Universal Robots PolyScope program: motion_capture.urp

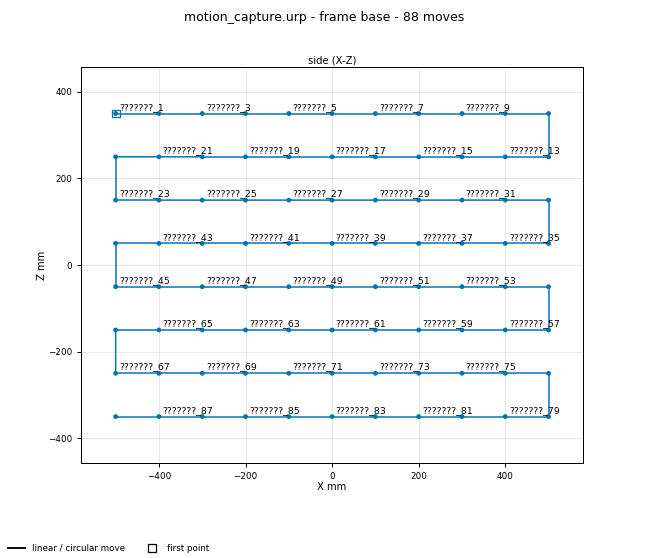
[picture p0: tool path of motion_capture.urp in frame base, 88 of 94 moves have a stored position in this frame; points joined in program order, loops and branches not executed]
Program motion_capture (installation=GD directory=/programs/GD createdIn=5.13.0 lastSavedIn=5.13.0 robotSerialNumber=20205000017)
Calibrated DH parameters: a=[-0.000157, -0.56303, -0.236706, -0.000074, -0.000109, 0]; d=[0.181705, 47.632387, 369.599619, -417.058513, 0.119878, 0.115667]; alpha=[1.570881, -0.005074, -0.001247, 1.56886, -1.570997, 0]; deltaTheta=[0, -0.405485, 5.544791, 1.143886, -0.000009, -0.000001]
InitVariablesNode
BeforeStart
  SuppressedNode
    Script file /programs/GD/ROVI/ROVI_RESET.script
      | def ROVI_RESET():
      |   if (not socket_open(host,port,socket_name)):
      |     rovi_err=902
      |     return False
      |   end
      |   socket_send_line("X0()",socket_name)
      |   ret=socket_read_line(socket_name,socket_timeout)
      |   if (ret == "OK"):
      |     rovi_err=0
      |   elif (ret == "NG"):
      |     rovi_err=to_num(socket_read_line(socket_name,socket_timeout))
      |   else:
      |     ret="NG"
      |     rovi_err=903
      |   end
      |   socket_close(socket_name)
      |   if (rovi_err != 0):
      |     if (is_popup):
      |       popup(str_cat(ret,rovi_err),title="X0",warning=True,blocking=True)
      |     end
      |     return False
      |   else:
      |     return True
      |   end
      | end
  SuppressedNode
    Script file /programs/GD/ROVI/ROVI_CAPTURE.script
      | def ROVI_CAPTURE():
      |   Y1=[0.0,0.0,0.0,0.0]
      | #  p=get_actual_tool_flange_pose()
      |   p=Bucket
      |   if (not socket_open(host,port,socket_name)):
      |     rovi_err=902
      |     return False
      |   end
      |   socket_send_string("X1(",socket_name)
      |   socket_send_string(p[0],socket_name)
      |   socket_send_string(",",socket_name)
      |   socket_send_string(p[1],socket_name)
      |   socket_send_string(",",socket_name)
      |   socket_send_string(p[2],socket_name)
      |   socket_send_string(",",socket_name)
      |   socket_send_string(p[3],socket_name)
      |   socket_send_string(",",socket_name)
      |   socket_send_string(p[4],socket_name)
      |   socket_send_string(",",socket_name)
      |   socket_send_string(p[5],socket_name)
      |   socket_send_line(")",socket_name)
      |   ret=socket_read_line(socket_name,socket_timeout)
      |   if (ret == "OK"):
      |     rovi_err=0
      |     f=socket_read_ascii_float(4,socket_name,socket_timeout)
      |     while (f[0]!=4):
      |       sleep(0.3)
      |       f=socket_read_ascii_float(4,socket_name,socket_timeout)
      |     end
      |     i=0
      |     while (i<4):
      |       Y1[i]=f[i+1]
      |       i=i+1
      |     end
      |   elif (ret == "NG"):
      |     rovi_err=to_num(socket_read_line(socket_name,socket_timeout))
      |   else:
      |     ret="NG"
      |     rovi_err=903
      |   end
      |   socket_close(socket_name)
      |   if (rovi_err != 0):
      |     if (is_popup):
      |       popup(str_cat(ret,rovi_err),title="X1",warning=True,blocking=True)
      |     end
      |     return False
      |   else:
      |     return True
      |   end
      | end
  SuppressedNode
    Script file /programs/GD/ROVI/ROVI_SOLVE.script
      | def ROVI_SOLVE(is_popup=is_popup):
      |   buf=p[10000.0,0.0,0.0,0.0,0.0,0.0]
      |   if (not socket_open(host,port,socket_name)):
      |     rovi_err=902
      |     return False
      |   end
      |   socket_send_line("X2()",socket_name)
      |   ret=socket_read_line(socket_name,socket_timeout)
      |   if (ret == "OK"):
      |     rovi_err=0
      |     f=socket_read_ascii_float(6,socket_name,socket_timeout)
      |     while (f[0]!=6):
      |       sleep(0.3)
      |       f=socket_read_ascii_float(6,socket_name,socket_timeout)
      |     end
      |     counter=0
      |     while (counter<6):
      |       buf[counter]=f[counter+1]
      |       counter=counter+1
      |     end
      |   elif (ret == "NG"):
      |     rovi_err=to_num(socket_read_line(socket_name,socket_timeout))
      |   else:
      |     ret="NG"
      |     rovi_err=903
      |   end
      |   sleep(1.0)
      |   socket_close(socket_name)
      |   if (rovi_err != 0):
      |     if (is_popup):
      |       popup(str_cat(ret,rovi_err),title="X2",warning=True,blocking=True)
      |     end
      |   end
      |   return buf
      | end
Robot Program (runOnlyOnce=true)
  SetPayload (workpieceName=k10)
  Set NoAction tcp=TCP_1
  MoveJ speed 30 deg/s, acceleration 10 deg/s^2 (useActiveTCP=true) feature=Base
    Waypoint Variable (Variable): variable(featureName=gHome_Position)
  Set NoAction tcp=TCP_RXF
  MoveL speed 150 mm/s, acceleration 50 mm/s^2 (useActiveTCP=true) feature=Base
    Waypoint Variable (Variable): variable(featureName=gGD_1_M_RXF)
    Wait Sleep waitTime=1
    Waypoint Variable (Variable): variable(featureName=gGD_1_LM_RXF)
    Wait Sleep waitTime=1
    Waypoint Variable (Variable): variable(featureName=gGD_1_RM_RXF)
    Wait Sleep waitTime=1
    Waypoint Variable (Variable): variable(featureName=gGD_1_M_RXF)
    Wait Sleep waitTime=1
  Set NoAction tcp=TCP_1
  MoveL speed 150 mm/s, acceleration 50 mm/s^2 (useActiveTCP=true) feature=Base
    Waypoint ウェイポイント_1: TCP in base x=-500 y=-769.756 z=350 mm, rx=0.0264 ry=3.1227 rz=0.1901 rad; joints [-109.516, -129.597, -26.308, -120.914, 88.133, -18.442] deg; TCP offset x=0 y=80 z=420 mm, rx=0 ry=0 rz=0 rad
    Wait Sleep waitTime=0.5
    Waypoint ウェイポイント_2: TCP in base x=-400 y=-769.779 z=350 mm, rx=0.0265 ry=3.1227 rz=0.1899 rad; joints [-104.117, -122.245, -38.613, -116.074, 88.811, -13.053] deg; TCP offset x=0 y=80 z=420 mm, rx=0 ry=0 rz=0 rad
    Wait Sleep waitTime=0.5
    Waypoint ウェイポイント_3: TCP in base x=-300 y=-769.79 z=350 mm, rx=0.0265 ry=3.1227 rz=0.19 rad; joints [-98.329, -117.36, -46.223, -113.407, 89.532, -7.291] deg; TCP offset x=0 y=80 z=420 mm, rx=0 ry=0 rz=0 rad
    Wait Sleep waitTime=0.5
    Waypoint ウェイポイント_4: TCP in base x=-200 y=-769.71 z=350 mm, rx=0.0266 ry=3.1227 rz=0.1902 rad; joints [-92.242, -114.037, -51.158, -111.783, 90.287, -1.234] deg; TCP offset x=0 y=80 z=420 mm, rx=0 ry=0 rz=0 rad
    Wait Sleep waitTime=0.5
    Waypoint ウェイポイント_5: TCP in base x=-100 y=-769.749 z=350 mm, rx=0.0265 ry=3.1226 rz=0.1902 rad; joints [-85.973, -112.05, -54.029, -110.799, 91.056, 4.991] deg; TCP offset x=0 y=80 z=420 mm, rx=0 ry=0 rz=0 rad
    Wait Sleep waitTime=0.5
    Waypoint ウェイポイント_6: TCP in base x=0 y=-769.753 z=350 mm, rx=0.0264 ry=3.1226 rz=0.1901 rad; joints [-79.663, -111.302, -55.123, -110.266, 91.808, 11.256] deg; TCP offset x=0 y=80 z=420 mm, rx=0 ry=0 rz=0 rad
    Wait Sleep waitTime=0.5
    Waypoint ウェイポイント_7: TCP in base x=100 y=-769.698 z=350 mm, rx=0.0267 ry=3.1226 rz=0.1903 rad; joints [-73.466, -111.79, -54.492, -110.156, 92.517, 17.424] deg; TCP offset x=0 y=80 z=420 mm, rx=0 ry=0 rz=0 rad
    Wait Sleep waitTime=0.5
    Waypoint ウェイポイント_8: TCP in base x=200 y=-769.721 z=350 mm, rx=0.0266 ry=3.1226 rz=0.1901 rad; joints [-67.519, -113.515, -52.099, -110.501, 93.157, 23.334] deg; TCP offset x=0 y=80 z=420 mm, rx=0 ry=0 rz=0 rad
    Wait Sleep waitTime=0.5
    Waypoint ウェイポイント_9: TCP in base x=300 y=-769.734 z=350 mm, rx=0.0266 ry=3.1226 rz=0.1901 rad; joints [-61.936, -116.543, -47.722, -111.491, 93.723, 28.888] deg; TCP offset x=0 y=80 z=420 mm, rx=0 ry=0 rz=0 rad
    Wait Sleep waitTime=0.5
    Waypoint ウェイポイント_10: TCP in base x=400 y=-769.744 z=350 mm, rx=0.0266 ry=3.1227 rz=0.1901 rad; joints [-56.783, -121.056, -40.852, -113.474, 94.202, 34.015] deg; TCP offset x=0 y=80 z=420 mm, rx=0 ry=0 rz=0 rad
    Wait Sleep waitTime=0.5
    Waypoint ウェイポイント_11: TCP in base x=500 y=-769.783 z=350 mm, rx=0.0265 ry=3.1227 rz=0.19 rad; joints [-52.094, -127.671, -30.053, -117.27, 94.603, 38.674] deg; TCP offset x=0 y=80 z=420 mm, rx=0 ry=0 rz=0 rad
    Wait Sleep waitTime=0.5
    Waypoint ウェイポイント_12: TCP in base x=500 y=-769.761 z=250 mm, rx=0.0265 ry=3.1227 rz=0.19 rad; joints [-52.14, -123.62, -47.179, -104.2, 94.621, 38.633] deg; TCP offset x=0 y=80 z=420 mm, rx=0 ry=0 rz=0 rad
    Wait Sleep waitTime=0.5
    Waypoint ウェイポイント_13: TCP in base x=400 y=-769.733 z=250 mm, rx=0.0265 ry=3.1226 rz=0.1902 rad; joints [-56.825, -118.405, -55.226, -101.754, 94.224, 33.97] deg; TCP offset x=0 y=80 z=420 mm, rx=0 ry=0 rz=0 rad
    Wait Sleep waitTime=0.5
    Waypoint ウェイポイント_14: TCP in base x=300 y=-769.78 z=250 mm, rx=0.0265 ry=3.1227 rz=0.1901 rad; joints [-61.971, -114.528, -60.888, -100.344, 93.735, 28.848] deg; TCP offset x=0 y=80 z=420 mm, rx=0 ry=0 rz=0 rad
    Wait Sleep waitTime=0.5
    Waypoint ウェイポイント_15: TCP in base x=200 y=-769.782 z=250 mm, rx=0.0265 ry=3.1227 rz=0.1902 rad; joints [-67.551, -111.827, -64.66, -99.633, 93.168, 23.296] deg; TCP offset x=0 y=80 z=420 mm, rx=0 ry=0 rz=0 rad
    Wait Sleep waitTime=0.5
    Waypoint ウェイポイント_16: TCP in base x=100 y=-769.767 z=250 mm, rx=0.0265 ry=3.1226 rz=0.19 rad; joints [-73.497, -110.242, -66.791, -99.399, 92.528, 17.384] deg; TCP offset x=0 y=80 z=420 mm, rx=0 ry=0 rz=0 rad
    Wait Sleep waitTime=0.5
    Waypoint ウェイポイント_17: TCP in base x=0 y=-769.774 z=250 mm, rx=0.0265 ry=3.1227 rz=0.1903 rad; joints [-79.694, -109.796, -67.348, -99.555, 91.819, 11.226] deg; TCP offset x=0 y=80 z=420 mm, rx=0 ry=0 rz=0 rad
    Wait Sleep waitTime=0.5
    Waypoint ウェイポイント_18: TCP in base x=-100 y=-769.761 z=250 mm, rx=0.0265 ry=3.1227 rz=0.1902 rad; joints [-86.003, -110.461, -66.398, -100.019, 91.066, 4.957] deg; TCP offset x=0 y=80 z=420 mm, rx=0 ry=0 rz=0 rad
    Wait Sleep waitTime=0.5
    Waypoint ウェイポイント_19: TCP in base x=-200 y=-769.774 z=250 mm, rx=0.0265 ry=3.1226 rz=0.19 rad; joints [-92.277, -112.252, -63.883, -100.838, 90.305, -1.28] deg; TCP offset x=0 y=80 z=420 mm, rx=0 ry=0 rz=0 rad
    Wait Sleep waitTime=0.5
    Waypoint ウェイポイント_20: TCP in base x=-300 y=-769.782 z=250 mm, rx=0.0266 ry=3.1227 rz=0.1902 rad; joints [-98.365, -115.185, -59.674, -102.136, 89.547, -7.327] deg; TCP offset x=0 y=80 z=420 mm, rx=0 ry=0 rz=0 rad
    Wait Sleep waitTime=0.5
    Waypoint ウェイポイント_21: TCP in base x=-400 y=-769.744 z=250.004 mm, rx=0.0265 ry=3.1226 rz=0.1902 rad; joints [-104.157, -119.31, -53.522, -104.109, 88.825, -13.094] deg; TCP offset x=0 y=80 z=420 mm, rx=0 ry=0 rz=0 rad
    Wait Sleep waitTime=0.5
    Waypoint ウェイポイント_22: TCP in base x=-500 y=-769.753 z=249.977 mm, rx=0.0265 ry=3.1226 rz=0.1903 rad; joints [-109.569, -124.862, -44.793, -107.171, 88.153, -18.483] deg; TCP offset x=0 y=80 z=420 mm, rx=0 ry=0 rz=0 rad
    Wait Sleep waitTime=0.5
    Waypoint ウェイポイント_23: TCP in base x=-500 y=-769.728 z=150 mm, rx=0.0264 ry=3.1227 rz=0.1902 rad; joints [-109.598, -123.814, -56.555, -96.452, 88.164, -18.521] deg; TCP offset x=0 y=80 z=420 mm, rx=0 ry=0 rz=0 rad
    Wait Sleep waitTime=0.5
    Waypoint ウェイポイント_24: TCP in base x=-400 y=-769.776 z=150 mm, rx=0.0265 ry=3.1226 rz=0.1901 rad; joints [-104.184, -118.927, -64.15, -93.858, 88.837, -13.124] deg; TCP offset x=0 y=80 z=420 mm, rx=0 ry=0 rz=0 rad
    Wait Sleep waitTime=0.5
    Waypoint ウェイポイント_25: TCP in base x=-300 y=-769.743 z=149.972 mm, rx=0.0267 ry=3.1226 rz=0.1901 rad; joints [-98.391, -115.168, -69.741, -92.084, 89.559, -7.356] deg; TCP offset x=0 y=80 z=420 mm, rx=0 ry=0 rz=0 rad
    Wait Sleep waitTime=0.5
    Waypoint ウェイポイント_26: TCP in base x=-200 y=-769.78 z=149.978 mm, rx=0.0265 ry=3.1226 rz=0.1901 rad; joints [-92.297, -112.457, -73.637, -90.88, 90.311, -1.304] deg; TCP offset x=0 y=80 z=420 mm, rx=0 ry=0 rz=0 rad
    Wait Sleep waitTime=0.5
    Waypoint ウェイポイント_27: TCP in base x=-100 y=-769.746 z=149.996 mm, rx=0.0265 ry=3.1226 rz=0.1901 rad; joints [-86.025, -110.779, -76.003, -90.094, 91.077, 4.925] deg; TCP offset x=0 y=80 z=420 mm, rx=0 ry=0 rz=0 rad
    Wait Sleep waitTime=0.5
    Waypoint ウェイポイント_28: TCP in base x=0 y=-769.794 z=149.992 mm, rx=0.0266 ry=3.1226 rz=0.19 rad; joints [-79.715, -110.158, -76.899, -89.634, 91.827, 11.198] deg; TCP offset x=0 y=80 z=420 mm, rx=0 ry=0 rz=0 rad
    Wait Sleep waitTime=0.5
    Waypoint ウェイポイント_29: TCP in base x=100 y=-769.807 z=149.986 mm, rx=0.0266 ry=3.1226 rz=0.1899 rad; joints [-73.519, -110.593, -76.354, -89.482, 92.536, 17.357] deg; TCP offset x=0 y=80 z=420 mm, rx=0 ry=0 rz=0 rad
    Wait Sleep waitTime=0.5
    Waypoint ウェイポイント_30: TCP in base x=200 y=-769.814 z=150.011 mm, rx=0.0265 ry=3.1226 rz=0.19 rad; joints [-67.576, -112.084, -74.34, -89.69, 93.18, 23.266] deg; TCP offset x=0 y=80 z=420 mm, rx=0 ry=0 rz=0 rad
    Wait Sleep waitTime=0.5
    Waypoint ウェイポイント_31: TCP in base x=300 y=-769.832 z=150.061 mm, rx=0.0265 ry=3.1227 rz=0.1899 rad; joints [-61.994, -114.608, -70.805, -90.341, 93.741, 28.822] deg; TCP offset x=0 y=80 z=420 mm, rx=0 ry=0 rz=0 rad
    Wait Sleep waitTime=0.5
    Waypoint ウェイポイント_32: TCP in base x=400 y=-769.796 z=150.029 mm, rx=0.0265 ry=3.1226 rz=0.19 rad; joints [-56.85, -118.168, -65.623, -91.587, 94.231, 33.94] deg; TCP offset x=0 y=80 z=420 mm, rx=0 ry=0 rz=0 rad
    Wait Sleep waitTime=0.5
    Waypoint ウェイポイント_33: TCP in base x=500 y=-769.794 z=150.02 mm, rx=0.0264 ry=3.1226 rz=0.19 rad; joints [-52.172, -122.824, -58.507, -93.665, 94.637, 38.595] deg; TCP offset x=0 y=80 z=420 mm, rx=0 ry=0 rz=0 rad
    Wait Sleep waitTime=0.5
    Waypoint ウェイポイント_34: TCP in base x=500 y=-769.78 z=50 mm, rx=0.0265 ry=3.1226 rz=0.1901 rad; joints [-52.19, -123.942, -66.82, -84.239, 94.645, 38.57] deg; TCP offset x=0 y=80 z=420 mm, rx=0 ry=0 rz=0 rad
    Wait Sleep waitTime=0.5
    Waypoint ウェイポイント_35: TCP in base x=400 y=-769.761 z=50 mm, rx=0.0265 ry=3.1226 rz=0.19 rad; joints [-56.865, -119.645, -73.521, -82.215, 94.236, 33.917] deg; TCP offset x=0 y=80 z=420 mm, rx=0 ry=0 rz=0 rad
    Wait Sleep waitTime=0.5
    Waypoint ウェイポイント_36: TCP in base x=300 y=-769.793 z=50 mm, rx=0.0264 ry=3.1227 rz=0.19 rad; joints [-62.007, -116.32, -78.49, -80.95, 93.746, 28.792] deg; TCP offset x=0 y=80 z=420 mm, rx=0 ry=0 rz=0 rad
    Wait Sleep waitTime=0.5
    Waypoint ウェイポイント_37: TCP in base x=200 y=-769.726 z=50 mm, rx=0.0266 ry=3.1227 rz=0.1901 rad; joints [-67.584, -113.935, -81.926, -80.261, 93.179, 23.251] deg; TCP offset x=0 y=80 z=420 mm, rx=0 ry=0 rz=0 rad
    Wait Sleep waitTime=0.5
    Waypoint ウェイポイント_38: TCP in base x=100 y=-769.734 z=50 mm, rx=0.0266 ry=3.1227 rz=0.1902 rad; joints [-73.528, -112.524, -83.891, -80.027, 92.535, 17.338] deg; TCP offset x=0 y=80 z=420 mm, rx=0 ry=0 rz=0 rad
    Wait Sleep waitTime=0.5
    Waypoint ウェイポイント_39: TCP in base x=0 y=-769.785 z=50 mm, rx=0.0265 ry=3.1227 rz=0.19 rad; joints [-79.723, -112.1, -84.439, -80.152, 91.823, 11.179] deg; TCP offset x=0 y=80 z=420 mm, rx=0 ry=0 rz=0 rad
    Wait Sleep waitTime=0.5
    Waypoint ウェイポイント_40: TCP in base x=-100 y=-769.765 z=50 mm, rx=0.0264 ry=3.1226 rz=0.1901 rad; joints [-86.037, -112.684, -83.567, -80.626, 91.077, 4.903] deg; TCP offset x=0 y=80 z=420 mm, rx=0 ry=0 rz=0 rad
    Wait Sleep waitTime=0.5
    Waypoint ウェイポイント_41: TCP in base x=-200 y=-769.713 z=50 mm, rx=0.0267 ry=3.1227 rz=0.1902 rad; joints [-92.31, -114.257, -81.273, -81.449, 90.311, -1.321] deg; TCP offset x=0 y=80 z=420 mm, rx=0 ry=0 rz=0 rad
    Wait Sleep waitTime=0.5
    Waypoint ウェイポイント_42: TCP in base x=-300 y=-769.709 z=50 mm, rx=0.0266 ry=3.1227 rz=0.1901 rad; joints [-98.402, -116.797, -77.512, -82.684, 89.556, -7.379] deg; TCP offset x=0 y=80 z=420 mm, rx=0 ry=0 rz=0 rad
    Wait Sleep waitTime=0.5
    Waypoint ウェイポイント_43: TCP in base x=-400 y=-769.724 z=50 mm, rx=0.0265 ry=3.1227 rz=0.1901 rad; joints [-104.199, -120.293, -72.183, -84.458, 88.839, -13.148] deg; TCP offset x=0 y=80 z=420 mm, rx=0 ry=0 rz=0 rad
    Wait Sleep waitTime=0.5
    Waypoint ウェイポイント_44: TCP in base x=-500 y=-769.745 z=50 mm, rx=0.0264 ry=3.1227 rz=0.1901 rad; joints [-109.616, -124.776, -65.087, -86.954, 88.17, -18.547] deg; TCP offset x=0 y=80 z=420 mm, rx=0 ry=0 rz=0 rad
    Wait Sleep waitTime=0.5
    Waypoint ウェイポイント_45: TCP in base x=-500 y=-769.748 z=-50 mm, rx=0.0265 ry=3.1226 rz=0.1901 rad; joints [-109.628, -127.262, -71.334, -78.222, 88.172, -18.572] deg; TCP offset x=0 y=80 z=420 mm, rx=0 ry=0 rz=0 rad
    Wait Sleep waitTime=0.5
    Waypoint ウェイポイント_46: TCP in base x=-400 y=-769.74 z=-50 mm, rx=0.0265 ry=3.1228 rz=0.1901 rad; joints [-104.206, -123.109, -78.194, -75.629, 88.834, -13.168] deg; TCP offset x=0 y=80 z=420 mm, rx=0 ry=0 rz=0 rad
    Wait Sleep waitTime=0.5
    Waypoint ウェイポイント_47: TCP in base x=-300 y=-769.776 z=-50 mm, rx=0.0264 ry=3.1227 rz=0.1901 rad; joints [-98.41, -119.861, -83.398, -73.732, 89.556, -7.407] deg; TCP offset x=0 y=80 z=420 mm, rx=0 ry=0 rz=0 rad
    Wait Sleep waitTime=0.5
    Waypoint ウェイポイント_48: TCP in base x=-200 y=-769.747 z=-50 mm, rx=0.0265 ry=3.1227 rz=0.1902 rad; joints [-92.317, -117.49, -87.11, -72.379, 90.309, -1.347] deg; TCP offset x=0 y=80 z=420 mm, rx=0 ry=0 rz=0 rad
    Wait Sleep waitTime=0.5
    Waypoint ウェイポイント_49: TCP in base x=-100 y=-769.782 z=-50 mm, rx=0.0265 ry=3.1226 rz=0.19 rad; joints [-86.045, -116.02, -89.387, -71.467, 91.076, 4.885] deg; TCP offset x=0 y=80 z=420 mm, rx=0 ry=0 rz=0 rad
    Wait Sleep waitTime=0.5
    Waypoint ウェイポイント_50: TCP in base x=0 y=-769.751 z=-50 mm, rx=0.0265 ry=3.1227 rz=0.19 rad; joints [-79.73, -115.477, -90.253, -70.961, 91.821, 11.159] deg; TCP offset x=0 y=80 z=420 mm, rx=0 ry=0 rz=0 rad
    Wait Sleep waitTime=0.5
    Waypoint ウェイポイント_51: TCP in base x=100 y=-769.758 z=-50 mm, rx=0.0264 ry=3.1226 rz=0.19 rad; joints [-73.536, -115.881, -89.7, -70.853, 92.534, 17.311] deg; TCP offset x=0 y=80 z=420 mm, rx=0 ry=0 rz=0 rad
    Wait Sleep waitTime=0.5
    Waypoint ウェイポイント_52: TCP in base x=200 y=-769.741 z=-50 mm, rx=0.0265 ry=3.1226 rz=0.19 rad; joints [-67.593, -117.213, -87.734, -71.173, 93.178, 23.224] deg; TCP offset x=0 y=80 z=420 mm, rx=0 ry=0 rz=0 rad
    Wait Sleep waitTime=0.5
    Waypoint ウェイポイント_53: TCP in base x=300 y=-769.771 z=-50 mm, rx=0.0264 ry=3.1227 rz=0.1901 rad; joints [-62.015, -119.452, -84.323, -71.99, 93.746, 28.773] deg; TCP offset x=0 y=80 z=420 mm, rx=0 ry=0 rz=0 rad
    Wait Sleep waitTime=0.5
    Waypoint ウェイポイント_54: TCP in base x=400 y=-769.796 z=-50 mm, rx=0.0265 ry=3.1226 rz=0.19 rad; joints [-56.874, -122.559, -79.436, -73.387, 94.233, 33.894] deg; TCP offset x=0 y=80 z=420 mm, rx=0 ry=0 rz=0 rad
    Wait Sleep waitTime=0.5
    Waypoint ウェイポイント_55: TCP in base x=500 y=-769.786 z=-50 mm, rx=0.0263 ry=3.1227 rz=0.1899 rad; joints [-52.197, -126.548, -72.935, -75.52, 94.64, 38.542] deg; TCP offset x=0 y=80 z=420 mm, rx=0 ry=0 rz=0 rad
    Wait Sleep waitTime=0.5
    Waypoint ウェイポイント_56: TCP in base x=500 y=-769.751 z=-150 mm, rx=0.0266 ry=3.1227 rz=0.19 rad; joints [-52.202, -130.42, -77.186, -67.402, 94.639, 38.529] deg; TCP offset x=0 y=80 z=420 mm, rx=0 ry=0 rz=0 rad
    Wait Sleep waitTime=0.5
    Waypoint ウェイポイント_57: TCP in base x=400 y=-769.754 z=-150 mm, rx=0.0264 ry=3.1227 rz=0.1902 rad; joints [-56.878, -126.74, -83.591, -65.064, 94.233, 33.868] deg; TCP offset x=0 y=80 z=420 mm, rx=0 ry=0 rz=0 rad
    Wait Sleep waitTime=0.5
    Waypoint ウェイポイント_58: TCP in base x=300 y=-769.728 z=-150 mm, rx=0.0264 ry=3.1227 rz=0.1901 rad; joints [-62.017, -123.86, -88.469, -63.437, 93.74, 28.754] deg; TCP offset x=0 y=80 z=420 mm, rx=0 ry=0 rz=0 rad
    Wait Sleep waitTime=0.5
    Waypoint ウェイポイント_59: TCP in base x=200 y=-769.736 z=-150 mm, rx=0.0265 ry=3.1227 rz=0.1901 rad; joints [-67.596, -121.798, -91.875, -62.45, 93.172, 23.205] deg; TCP offset x=0 y=80 z=420 mm, rx=0 ry=0 rz=0 rad
    Wait Sleep waitTime=0.5
    Waypoint ウェイポイント_60: TCP in base x=100 y=-769.719 z=-150 mm, rx=0.0265 ry=3.1227 rz=0.19 rad; joints [-73.536, -120.562, -93.861, -62.015, 92.523, 17.299] deg; TCP offset x=0 y=80 z=420 mm, rx=0 ry=0 rz=0 rad
    Wait Sleep waitTime=0.5
    Waypoint ウェイポイント_61: TCP in base x=0 y=-769.761 z=-150 mm, rx=0.0265 ry=3.1227 rz=0.1901 rad; joints [-79.735, -120.19, -94.412, -62.094, 91.818, 11.136] deg; TCP offset x=0 y=80 z=420 mm, rx=0 ry=0 rz=0 rad
    Wait Sleep waitTime=0.5
    Waypoint ウェイポイント_62: TCP in base x=-100 y=-769.768 z=-150 mm, rx=0.0265 ry=3.1227 rz=0.1899 rad; joints [-86.045, -120.674, -93.563, -62.634, 91.064, 4.869] deg; TCP offset x=0 y=80 z=420 mm, rx=0 ry=0 rz=0 rad
    Wait Sleep waitTime=0.5
    Waypoint ウェイポイント_63: TCP in base x=-200 y=-769.762 z=-150 mm, rx=0.0266 ry=3.1227 rz=0.19 rad; joints [-92.319, -122.018, -91.291, -63.662, 90.301, -1.365] deg; TCP offset x=0 y=80 z=420 mm, rx=0 ry=0 rz=0 rad
    Wait Sleep waitTime=0.5
    Waypoint ウェイポイント_64: TCP in base x=-300 y=-769.778 z=-150 mm, rx=0.0265 ry=3.1226 rz=0.19 rad; joints [-98.416, -124.201, -87.585, -65.203, 89.554, -7.427] deg; TCP offset x=0 y=80 z=420 mm, rx=0 ry=0 rz=0 rad
    Wait Sleep waitTime=0.5
    Waypoint ウェイポイント_65: TCP in base x=-400 y=-769.718 z=-150 mm, rx=0.0266 ry=3.1227 rz=0.1901 rad; joints [-104.214, -127.194, -82.425, -67.314, 88.835, -13.191] deg; TCP offset x=0 y=80 z=420 mm, rx=0 ry=0 rz=0 rad
    Wait Sleep waitTime=0.5
    Waypoint ウェイポイント_66: TCP in base x=-500 y=-769.745 z=-150 mm, rx=0.0266 ry=3.1226 rz=0.1901 rad; joints [-109.636, -131.024, -75.681, -70.112, 88.172, -18.591] deg; TCP offset x=0 y=80 z=420 mm, rx=0 ry=0 rz=0 rad
    Wait Sleep waitTime=0.5
    Waypoint ウェイポイント_67: TCP in base x=-500.003 y=-769.738 z=-250 mm, rx=0.0266 ry=3.1227 rz=0.19 rad; joints [-109.638, -135.891, -78.285, -62.637, 88.168, -18.615] deg; TCP offset x=0 y=80 z=420 mm, rx=0 ry=0 rz=0 rad
    Wait Sleep waitTime=0.5
    Waypoint ウェイポイント_68: TCP in base x=-400 y=-769.765 z=-250 mm, rx=0.0265 ry=3.1227 rz=0.19 rad; joints [-104.213, -132.393, -84.974, -59.563, 88.827, -13.214] deg; TCP offset x=0 y=80 z=420 mm, rx=0 ry=0 rz=0 rad
    Wait Sleep waitTime=0.5
    Waypoint ウェイポイント_69: TCP in base x=-300 y=-769.757 z=-250 mm, rx=0.0265 ry=3.1226 rz=0.1901 rad; joints [-98.417, -129.68, -90.119, -57.196, 89.546, -7.448] deg; TCP offset x=0 y=80 z=420 mm, rx=0 ry=0 rz=0 rad
    Wait Sleep waitTime=0.5
    Waypoint ウェイポイント_70: TCP in base x=-200 y=-769.86 z=-250 mm, rx=0.0266 ry=3.1226 rz=0.1899 rad; joints [-92.323, -127.719, -93.818, -55.431, 90.298, -1.389] deg; TCP offset x=0 y=80 z=420 mm, rx=0 ry=0 rz=0 rad
    Wait Sleep waitTime=0.5
    Waypoint ウェイポイント_71: TCP in base x=-100 y=-769.753 z=-250 mm, rx=0.0266 ry=3.1226 rz=0.19 rad; joints [-86.048, -126.514, -96.102, -54.258, 91.061, 4.845] deg; TCP offset x=0 y=80 z=420 mm, rx=0 ry=0 rz=0 rad
    Wait Sleep waitTime=0.5
    Waypoint ウェイポイント_72: TCP in base x=0 y=-769.75 z=-250 mm, rx=0.0265 ry=3.1227 rz=0.19 rad; joints [-79.735, -126.084, -96.958, -53.651, 91.808, 11.116] deg; TCP offset x=0 y=80 z=420 mm, rx=0 ry=0 rz=0 rad
    Wait Sleep waitTime=0.5
    Waypoint ウェイポイント_73: TCP in base x=100 y=-769.75 z=-250 mm, rx=0.0266 ry=3.1227 rz=0.19 rad; joints [-73.538, -126.43, -96.384, -53.624, 92.517, 17.278] deg; TCP offset x=0 y=80 z=420 mm, rx=0 ry=0 rz=0 rad
    Wait Sleep waitTime=0.5
    Waypoint ウェイポイント_74: TCP in base x=200 y=-769.767 z=-250 mm, rx=0.0266 ry=3.1226 rz=0.1901 rad; joints [-67.601, -127.547, -94.381, -54.196, 93.17, 23.181] deg; TCP offset x=0 y=80 z=420 mm, rx=0 ry=0 rz=0 rad
    Wait Sleep waitTime=0.5
    Waypoint ウェイポイント_75: TCP in base x=300 y=-769.739 z=-250 mm, rx=0.0265 ry=3.1227 rz=0.19 rad; joints [-62.018, -129.409, -90.965, -55.392, 93.733, 28.734] deg; TCP offset x=0 y=80 z=420 mm, rx=0 ry=0 rz=0 rad
    Wait Sleep waitTime=0.5
    Waypoint ウェイポイント_76: TCP in base x=400 y=-769.737 z=-250 mm, rx=0.0266 ry=3.1227 rz=0.1901 rad; joints [-56.878, -132.022, -86.092, -57.278, 94.226, 33.852] deg; TCP offset x=0 y=80 z=420 mm, rx=0 ry=0 rz=0 rad
    Wait Sleep waitTime=0.5
    Waypoint ウェイポイント_77: TCP in base x=500 y=-769.789 z=-250 mm, rx=0.0265 ry=3.1227 rz=0.1901 rad; joints [-52.205, -135.398, -79.696, -59.918, 94.635, 38.5] deg; TCP offset x=0 y=80 z=420 mm, rx=0 ry=0 rz=0 rad
    Wait Sleep waitTime=0.5
    Waypoint ウェイポイント_78: TCP in base x=500 y=-769.746 z=-350 mm, rx=0.0266 ry=3.1226 rz=0.19 rad; joints [-52.204, -141.306, -80.553, -53.152, 94.635, 38.481] deg; TCP offset x=0 y=80 z=420 mm, rx=0 ry=0 rz=0 rad
    Wait Sleep waitTime=0.5
    Waypoint ウェイポイント_79: TCP in base x=400 y=-769.754 z=-350 mm, rx=0.0265 ry=3.1227 rz=0.1901 rad; joints [-56.877, -138.256, -86.938, -50.197, 94.22, 33.823] deg; TCP offset x=0 y=80 z=420 mm, rx=0 ry=0 rz=0 rad
    Wait Sleep waitTime=0.5
    Waypoint ウェイポイント_80: TCP in base x=300 y=-769.759 z=-350 mm, rx=0.0265 ry=3.1227 rz=0.19 rad; joints [-62.017, -135.921, -91.823, -48.021, 93.726, 28.708] deg; TCP offset x=0 y=80 z=420 mm, rx=0 ry=0 rz=0 rad
    Wait Sleep waitTime=0.5
    Waypoint ウェイポイント_81: TCP in base x=200 y=-769.782 z=-350 mm, rx=0.0265 ry=3.1227 rz=0.1901 rad; joints [-67.594, -134.274, -95.253, -46.599, 93.154, 23.156] deg; TCP offset x=0 y=80 z=420 mm, rx=0 ry=0 rz=0 rad
    Wait Sleep waitTime=0.5
    Waypoint ウェイポイント_82: TCP in base x=100 y=-769.77 z=-350 mm, rx=0.0265 ry=3.1226 rz=0.1902 rad; joints [-73.539, -133.295, -97.262, -45.886, 92.511, 17.247] deg; TCP offset x=0 y=80 z=420 mm, rx=0 ry=0 rz=0 rad
    Wait Sleep waitTime=0.5
    Waypoint ウェイポイント_83: TCP in base x=0 y=-769.732 z=-350 mm, rx=0.0265 ry=3.1227 rz=0.1901 rad; joints [-79.733, -132.983, -97.851, -45.864, 91.798, 11.091] deg; TCP offset x=0 y=80 z=420 mm, rx=0 ry=0 rz=0 rad
    Wait Sleep waitTime=0.5
    Waypoint ウェイポイント_84: TCP in base x=-100 y=-769.749 z=-350 mm, rx=0.0264 ry=3.1227 rz=0.19 rad; joints [-86.043, -133.347, -97.005, -46.524, 91.048, 4.819] deg; TCP offset x=0 y=80 z=420 mm, rx=0 ry=0 rz=0 rad
    Wait Sleep waitTime=0.5
    Waypoint ウェイポイント_85: TCP in base x=-200 y=-769.743 z=-350 mm, rx=0.0265 ry=3.1227 rz=0.1901 rad; joints [-92.32, -134.391, -94.728, -47.856, 90.287, -1.415] deg; TCP offset x=0 y=80 z=420 mm, rx=0 ry=0 rz=0 rad
    Wait Sleep waitTime=0.5
    Waypoint ウェイポイント_86: TCP in base x=-300 y=-769.789 z=-350 mm, rx=0.0266 ry=3.1226 rz=0.1901 rad; joints [-98.416, -136.121, -91.018, -49.852, 89.539, -7.472] deg; TCP offset x=0 y=80 z=420 mm, rx=0 ry=0 rz=0 rad
    Wait Sleep waitTime=0.5
    Waypoint ウェイポイント_87: TCP in base x=-400 y=-769.751 z=-350 mm, rx=0.0266 ry=3.1226 rz=0.1901 rad; joints [-104.216, -138.546, -85.866, -52.524, 88.828, -13.24] deg; TCP offset x=0 y=80 z=420 mm, rx=0 ry=0 rz=0 rad
    Wait Sleep waitTime=0.5
    Waypoint ウェイポイント_88: TCP in base x=-500 y=-769.691 z=-350 mm, rx=0.0266 ry=3.1227 rz=0.1902 rad; joints [-109.636, -141.71, -79.193, -55.916, 88.161, -18.64] deg; TCP offset x=0 y=80 z=420 mm, rx=0 ry=0 rz=0 rad
    Wait Sleep waitTime=0.5
    MoveJ speed 30 deg/s, acceleration 10 deg/s^2 (useActiveTCP=true) feature=Base
      Waypoint Variable (Variable): variable(featureName=gHome_Position)
    Halt
